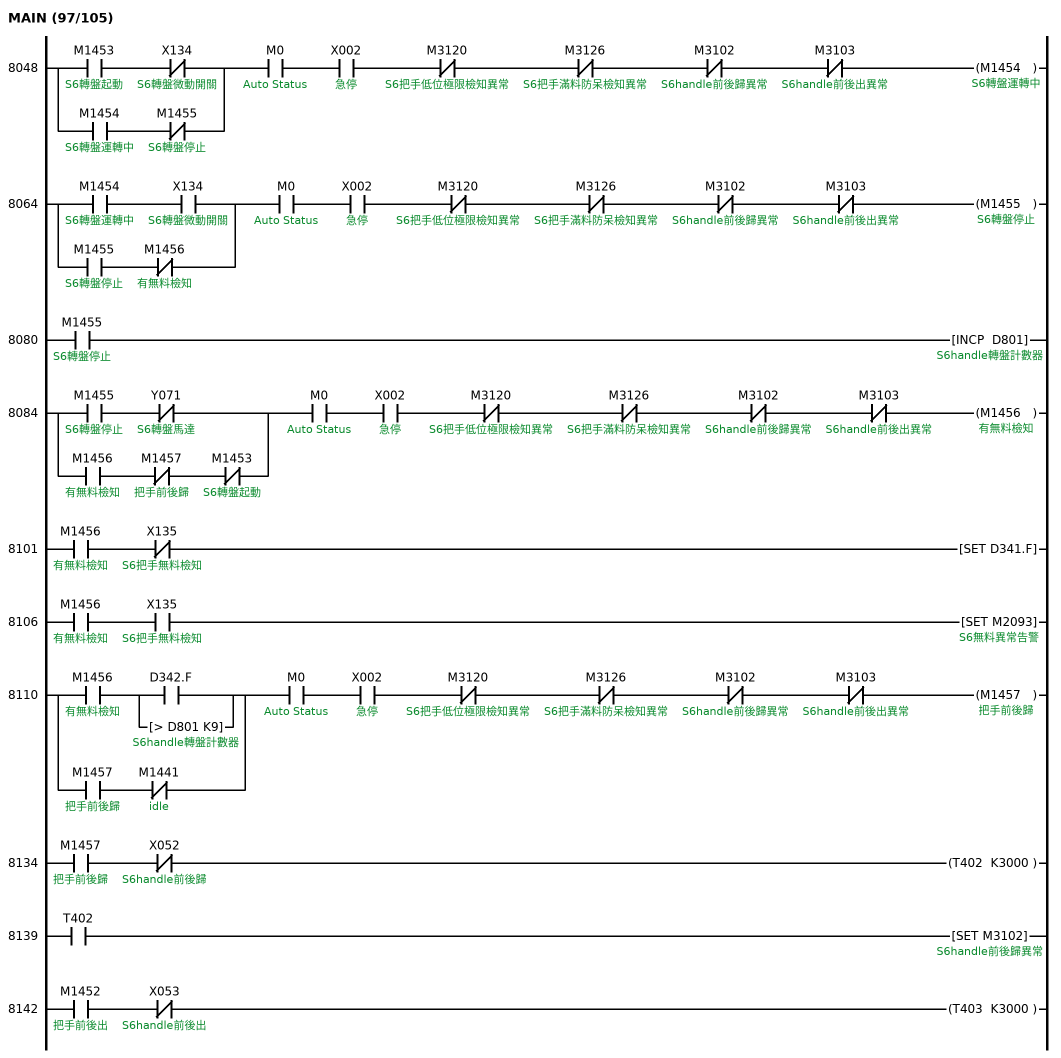
[picture p96: ladder of MAIN, rungs at steps 8048 to 8142]
8048  LD      M1453  ; S6轉盤起動
      ANI     X134  ; S6轉盤微動開關
      LD      M1454  ; S6轉盤運轉中
      ANI     M1455  ; S6轉盤停止
      ORB
      AND     M0  ; Auto Status
      AND     X002  ; 急停
      ANI     M3120  ; S6把手低位極限檢知異常
      ANI     M3126  ; S6把手滿料防呆檢知異常
      ANI     M3102  ; S6handle前後歸異常
      ANI     M3103  ; S6handle前後出異常
      OUT     M1454  ; S6轉盤運轉中
8064  LD      M1454  ; S6轉盤運轉中
      AND     X134  ; S6轉盤微動開關
      LD      M1455  ; S6轉盤停止
      ANI     M1456  ; 有無料檢知
      ORB
      AND     M0  ; Auto Status
      AND     X002  ; 急停
      ANI     M3120  ; S6把手低位極限檢知異常
      ANI     M3126  ; S6把手滿料防呆檢知異常
      ANI     M3102  ; S6handle前後歸異常
      ANI     M3103  ; S6handle前後出異常
      OUT     M1455  ; S6轉盤停止
8080  LD      M1455  ; S6轉盤停止
      INCP    D801
8084  LD      M1455  ; S6轉盤停止
      ANI     Y071  ; S6轉盤馬達
      LD      M1456  ; 有無料檢知
      ANI     M1457  ; 把手前後歸
      ANI     M1453  ; S6轉盤起動
      ORB
      AND     M0  ; Auto Status
      AND     X002  ; 急停
      ANI     M3120  ; S6把手低位極限檢知異常
      ANI     M3126  ; S6把手滿料防呆檢知異常
      ANI     M3102  ; S6handle前後歸異常
      ANI     M3103  ; S6handle前後出異常
      OUT     M1456  ; 有無料檢知
8101  LD      M1456  ; 有無料檢知
      ANI     X135  ; S6把手無料檢知
      SET     D341.F
8106  LD      M1456  ; 有無料檢知
      AND     X135  ; S6把手無料檢知
      SET     M2093  ; S6無料異常告警
8110  LD      M1456  ; 有無料檢知
      LD      D342.F
      OR>     D801 K9  ; S6handle轉盤計數器
      ANB
      LD      M1457  ; 把手前後歸
      ANI     M1441  ; idle
      ORB
      AND     M0  ; Auto Status
      AND     X002  ; 急停
      ANI     M3120  ; S6把手低位極限檢知異常
      ANI     M3126  ; S6把手滿料防呆檢知異常
      ANI     M3102  ; S6handle前後歸異常
      ANI     M3103  ; S6handle前後出異常
      OUT     M1457  ; 把手前後歸
8134  LD      M1457  ; 把手前後歸
      ANI     X052  ; S6handle前後歸
      OUT     T402 K3000
8139  LD      T402
      SET     M3102  ; S6handle前後歸異常
8142  LD      M1452  ; 把手前後出
      ANI     X053  ; S6handle前後出
      OUT     T403 K3000
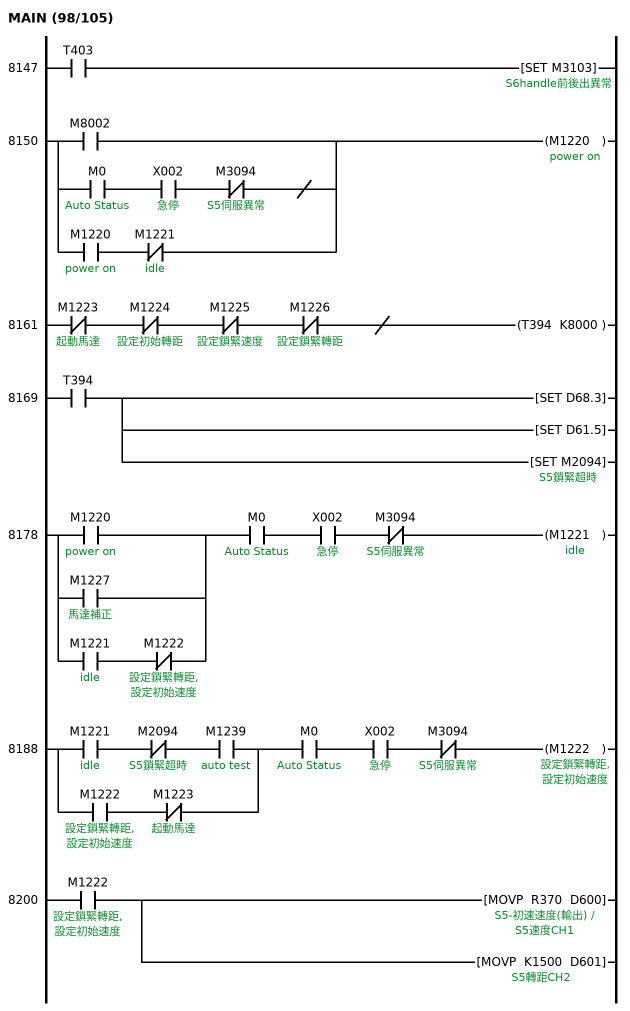
8147  LD      T403
      SET     M3103  ; S6handle前後出異常
8150  LD      M8002
      LD      M0  ; Auto Status
      AND     X002  ; 急停
      ANI     M3094  ; S5伺服異常
      INV
      ORB
      LD      M1220  ; power on
      ANI     M1221  ; idle
      ORB
      OUT     M1220  ; power on
8161  LDI     M1223  ; 起動馬達
      ANI     M1224  ; 設定初始轉距
      ANI     M1225  ; 設定鎖緊速度
      ANI     M1226  ; 設定鎖緊轉距
      INV
      OUT     T394 K8000
8169  LD      T394
      SET     D68.3
      SET     D61.5
      SET     M2094  ; S5鎖緊超時
8178  LD      M1220  ; power on
      OR      M1227  ; 馬達補正
      LD      M1221  ; idle
      ANI     M1222  ; 設定鎖緊轉距,設定初始速度
      ORB
      AND     M0  ; Auto Status
      AND     X002  ; 急停
      ANI     M3094  ; S5伺服異常
      OUT     M1221  ; idle
8188  LD      M1221  ; idle
      ANI     M2094  ; S5鎖緊超時
      AND     M1239  ; auto test
      LD      M1222  ; 設定鎖緊轉距,設定初始速度
      ANI     M1223  ; 起動馬達
      ORB
      AND     M0  ; Auto Status
      AND     X002  ; 急停
      ANI     M3094  ; S5伺服異常
      OUT     M1222  ; 設定鎖緊轉距,設定初始速度
8200  LD      M1222  ; 設定鎖緊轉距,設定初始速度
      MOVP    R370 D600
      MOVP    K1500 D601  ; S5轉距CH2
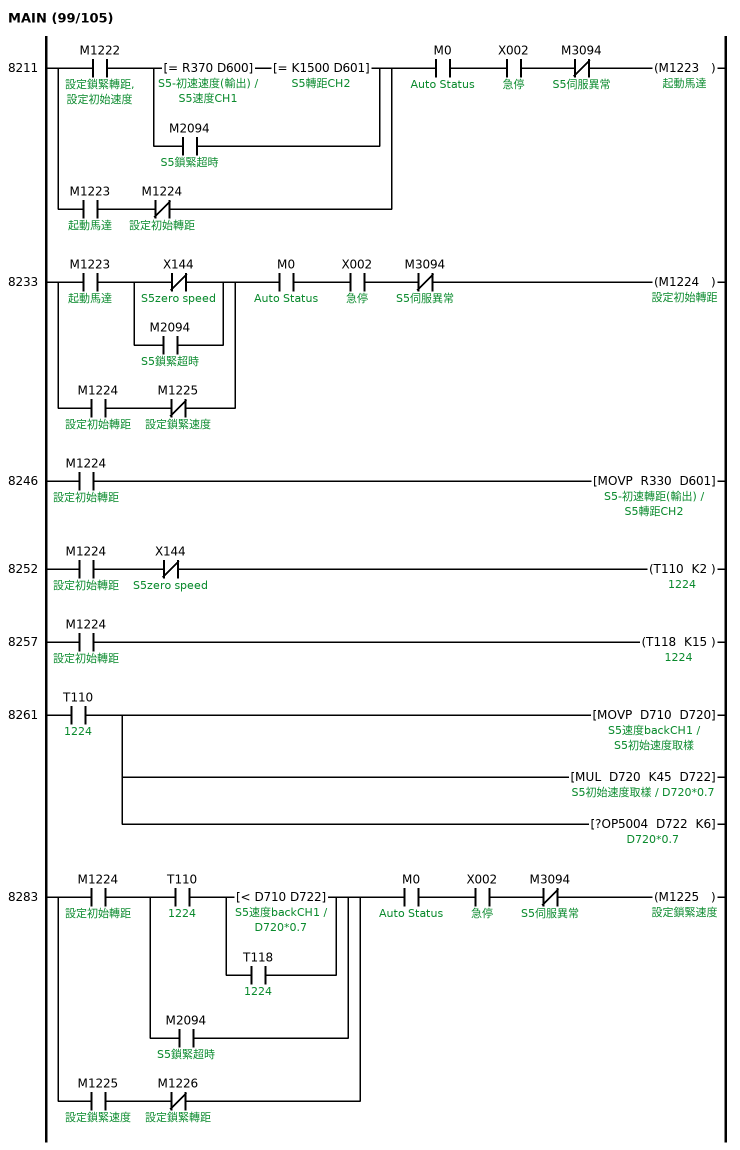
8211  LD      M1222  ; 設定鎖緊轉距,設定初始速度
      LD=     R370 D600  ; S5-初速速度(輸出) / S5速度CH1
      AND=    K1500 D601  ; S5轉距CH2
      OR      M2094  ; S5鎖緊超時
      ANB
      LD      M1223  ; 起動馬達
      ANI     M1224  ; 設定初始轉距
      ORB
      AND     M0  ; Auto Status
      AND     X002  ; 急停
      ANI     M3094  ; S5伺服異常
      OUT     M1223  ; 起動馬達
8233  LD      M1223  ; 起動馬達
      LDI     X144  ; S5zero speed
      OR      M2094  ; S5鎖緊超時
      ANB
      LD      M1224  ; 設定初始轉距
      ANI     M1225  ; 設定鎖緊速度
      ORB
      AND     M0  ; Auto Status
      AND     X002  ; 急停
      ANI     M3094  ; S5伺服異常
      OUT     M1224  ; 設定初始轉距
8246  LD      M1224  ; 設定初始轉距
      MOVP    R330 D601
8252  LD      M1224  ; 設定初始轉距
      ANI     X144  ; S5zero speed
      OUT     T110 K2  ; 1224
8257  LD      M1224  ; 設定初始轉距
      OUT     T118 K15  ; 1224
8261  LD      T110  ; 1224
      MOVP    D710 D720  ; S5初始速度取樣
      MUL     D720 K45 D722  ; D720*0.7
      ?OP5004 D722 K6
8283  LD      M1224  ; 設定初始轉距
      LD      T110  ; 1224
      LD<     D710 D722  ; S5速度backCH1 / D720*0.7
      OR      T118  ; 1224
      ANB
      OR      M2094  ; S5鎖緊超時
      ANB
      LD      M1225  ; 設定鎖緊速度
      ANI     M1226  ; 設定鎖緊轉距
      ORB
      AND     M0  ; Auto Status
      AND     X002  ; 急停
      ANI     M3094  ; S5伺服異常
      OUT     M1225  ; 設定鎖緊速度
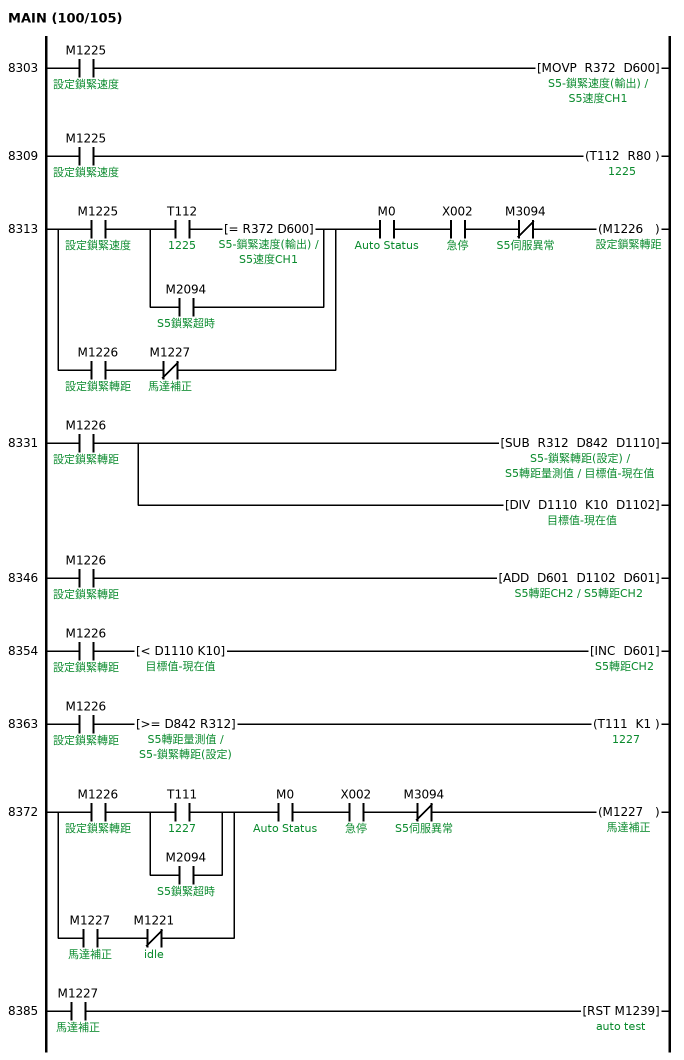
8303  LD      M1225  ; 設定鎖緊速度
      MOVP    R372 D600
8309  LD      M1225  ; 設定鎖緊速度
      OUT     T112 R80  ; 1225
8313  LD      M1225  ; 設定鎖緊速度
      LD      T112  ; 1225
      AND=    R372 D600  ; S5-鎖緊速度(輸出) / S5速度CH1
      OR      M2094  ; S5鎖緊超時
      ANB
      LD      M1226  ; 設定鎖緊轉距
      ANI     M1227  ; 馬達補正
      ORB
      AND     M0  ; Auto Status
      AND     X002  ; 急停
      ANI     M3094  ; S5伺服異常
      OUT     M1226  ; 設定鎖緊轉距
8331  LD      M1226  ; 設定鎖緊轉距
      SUB     R312 D842 D1110  ; 目標值-現在值
      DIV     D1110 K10 D1102
8346  LD      M1226  ; 設定鎖緊轉距
      ADD     D601 D1102 D601
8354  LD      M1226  ; 設定鎖緊轉距
      AND<    D1110 K10  ; 目標值-現在值
      INC     D601
8363  LD      M1226  ; 設定鎖緊轉距
      AND>=   D842 R312  ; S5轉距量測值 / S5-鎖緊轉距(設定)
      OUT     T111 K1  ; 1227
8372  LD      M1226  ; 設定鎖緊轉距
      LD      T111  ; 1227
      OR      M2094  ; S5鎖緊超時
      ANB
      LD      M1227  ; 馬達補正
      ANI     M1221  ; idle
      ORB
      AND     M0  ; Auto Status
      AND     X002  ; 急停
      ANI     M3094  ; S5伺服異常
      OUT     M1227  ; 馬達補正
8385  LD      M1227  ; 馬達補正
      RST     M1239  ; auto test
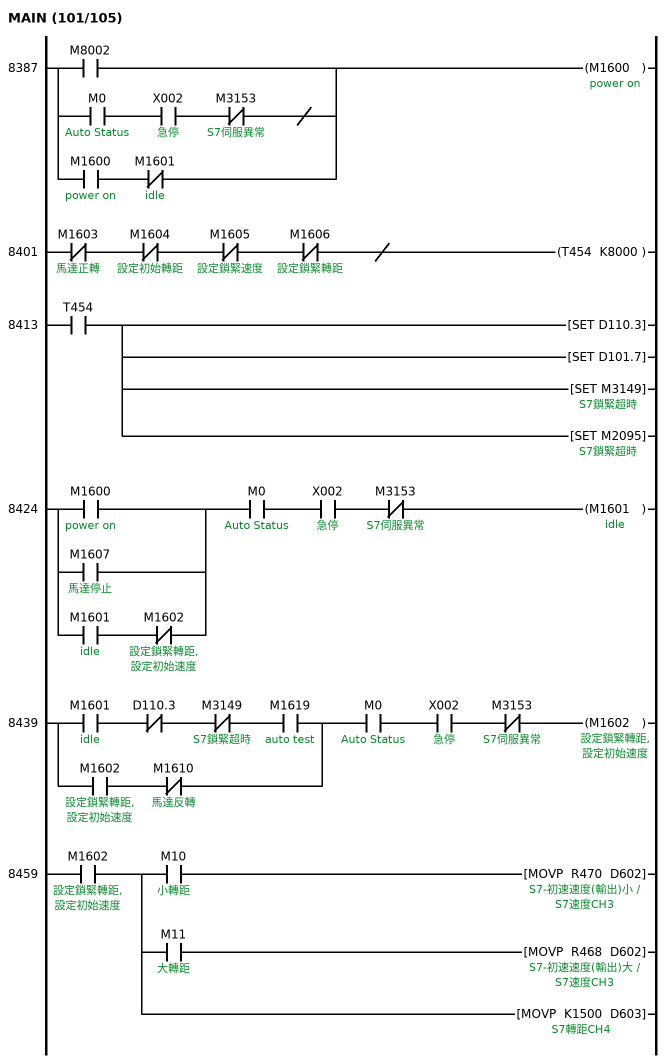
8387  LD      M8002
      LD      M0  ; Auto Status
      AND     X002  ; 急停
      ANI     M3153  ; S7伺服異常
      INV
      ORB
      LD      M1600  ; power on
      ANI     M1601  ; idle
      ORB
      OUT     M1600  ; power on
8401  LDI     M1603  ; 馬達正轉
      ANI     M1604  ; 設定初始轉距
      ANI     M1605  ; 設定鎖緊速度
      ANI     M1606  ; 設定鎖緊轉距
      INV
      OUT     T454 K8000
8413  LD      T454
      SET     D110.3
      SET     D101.7
      SET     M3149  ; S7鎖緊超時
      SET     M2095  ; S7鎖緊超時
8424  LD      M1600  ; power on
      OR      M1607  ; 馬達停止
      LD      M1601  ; idle
      ANI     M1602  ; 設定鎖緊轉距,設定初始速度
      ORB
      AND     M0  ; Auto Status
      AND     X002  ; 急停
      ANI     M3153  ; S7伺服異常
      OUT     M1601  ; idle
8439  LD      M1601  ; idle
      ANI     D110.3
      ANI     M3149  ; S7鎖緊超時
      AND     M1619  ; auto test
      LD      M1602  ; 設定鎖緊轉距,設定初始速度
      ANI     M1610  ; 馬達反轉
      ORB
      AND     M0  ; Auto Status
      AND     X002  ; 急停
      ANI     M3153  ; S7伺服異常
      OUT     M1602  ; 設定鎖緊轉距,設定初始速度
8459  LD      M1602  ; 設定鎖緊轉距,設定初始速度
      MPS
      AND     M10  ; 小轉距
      MOVP    R470 D602
      MRD
      AND     M11  ; 大轉距
      MOVP    R468 D602
      MPP
      MOVP    K1500 D603
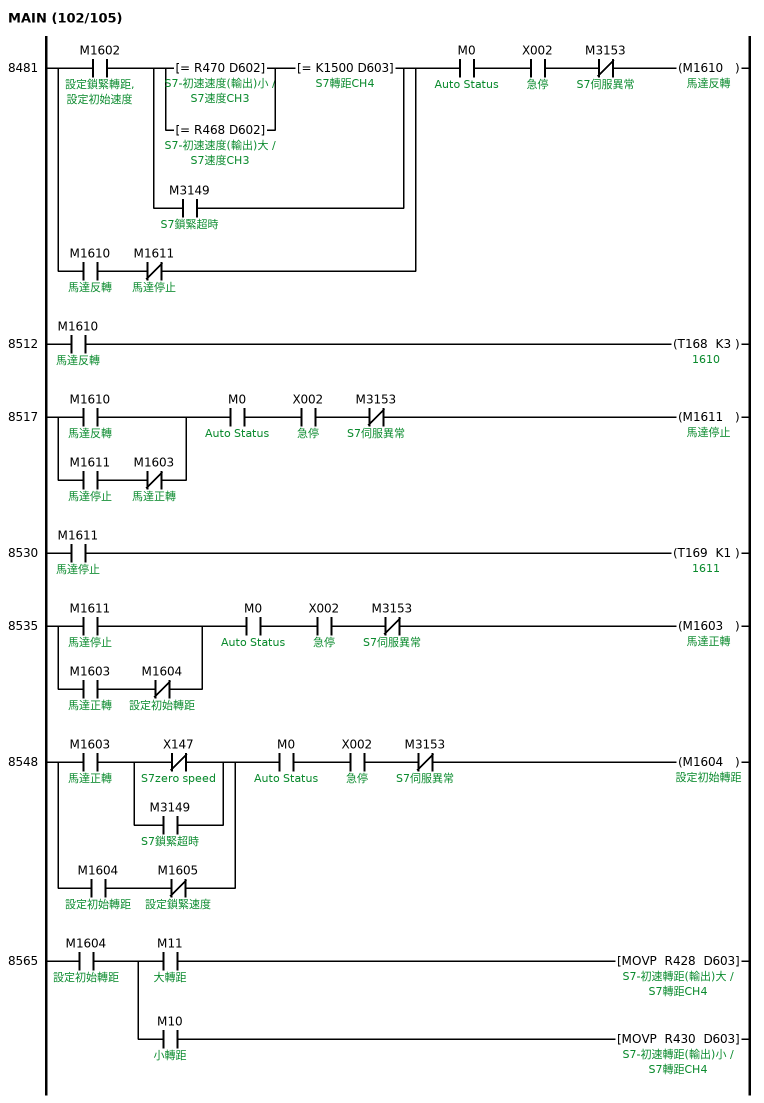
8481  LD      M1602  ; 設定鎖緊轉距,設定初始速度
      LD=     R470 D602  ; S7-初速速度(輸出)小 / S7速度CH3
      OR=     R468 D602  ; S7-初速速度(輸出)大 / S7速度CH3
      AND=    K1500 D603  ; S7轉距CH4
      OR      M3149  ; S7鎖緊超時
      ANB
      LD      M1610  ; 馬達反轉
      ANI     M1611  ; 馬達停止
      ORB
      AND     M0  ; Auto Status
      AND     X002  ; 急停
      ANI     M3153  ; S7伺服異常
      OUT     M1610  ; 馬達反轉
8512  LD      M1610  ; 馬達反轉
      OUT     T168 K3  ; 1610
8517  LD      M1610  ; 馬達反轉
      LD      M1611  ; 馬達停止
      ANI     M1603  ; 馬達正轉
      ORB
      AND     M0  ; Auto Status
      AND     X002  ; 急停
      ANI     M3153  ; S7伺服異常
      OUT     M1611  ; 馬達停止
8530  LD      M1611  ; 馬達停止
      OUT     T169 K1  ; 1611
8535  LD      M1611  ; 馬達停止
      LD      M1603  ; 馬達正轉
      ANI     M1604  ; 設定初始轉距
      ORB
      AND     M0  ; Auto Status
      AND     X002  ; 急停
      ANI     M3153  ; S7伺服異常
      OUT     M1603  ; 馬達正轉
8548  LD      M1603  ; 馬達正轉
      LDI     X147  ; S7zero speed
      OR      M3149  ; S7鎖緊超時
      ANB
      LD      M1604  ; 設定初始轉距
      ANI     M1605  ; 設定鎖緊速度
      ORB
      AND     M0  ; Auto Status
      AND     X002  ; 急停
      ANI     M3153  ; S7伺服異常
      OUT     M1604  ; 設定初始轉距
8565  LD      M1604  ; 設定初始轉距
      MPS
      AND     M11  ; 大轉距
      MOVP    R428 D603
      MPP
      AND     M10  ; 小轉距
      MOVP    R430 D603
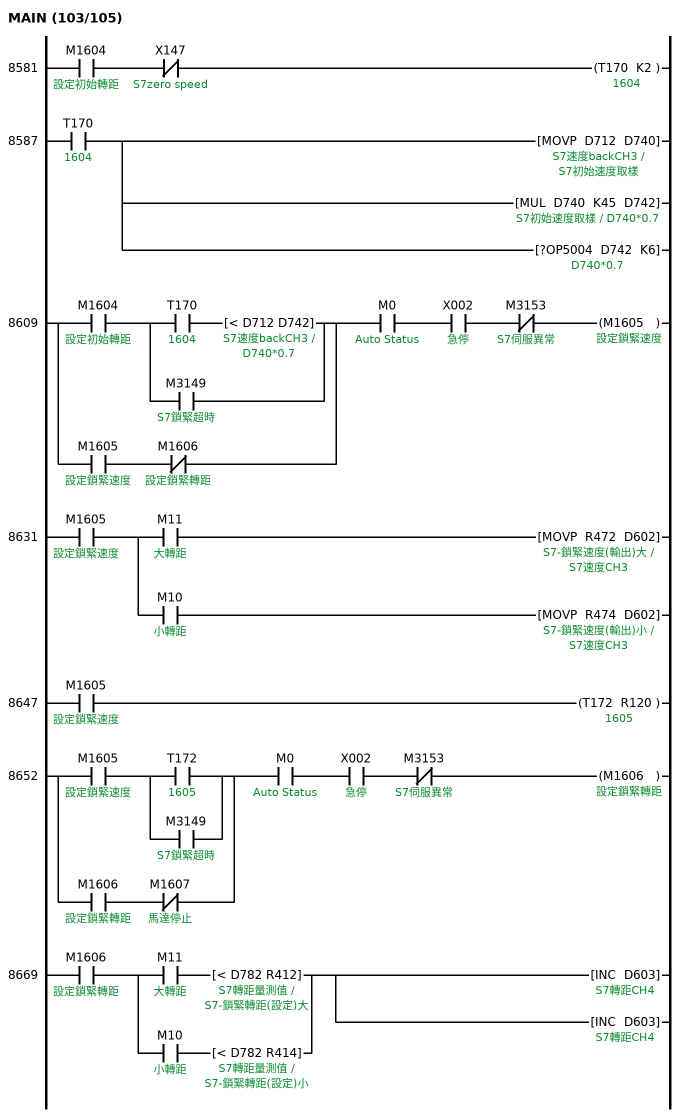
8581  LD      M1604  ; 設定初始轉距
      ANI     X147  ; S7zero speed
      OUT     T170 K2  ; 1604
8587  LD      T170  ; 1604
      MOVP    D712 D740  ; S7速度backCH3 / S7初始速度取樣
      MUL     D740 K45 D742  ; D740*0.7
      ?OP5004 D742 K6
8609  LD      M1604  ; 設定初始轉距
      LD      T170  ; 1604
      AND<    D712 D742  ; S7速度backCH3 / D740*0.7
      OR      M3149  ; S7鎖緊超時
      ANB
      LD      M1605  ; 設定鎖緊速度
      ANI     M1606  ; 設定鎖緊轉距
      ORB
      AND     M0  ; Auto Status
      AND     X002  ; 急停
      ANI     M3153  ; S7伺服異常
      OUT     M1605  ; 設定鎖緊速度
8631  LD      M1605  ; 設定鎖緊速度
      MPS
      AND     M11  ; 大轉距
      MOVP    R472 D602
      MPP
      AND     M10  ; 小轉距
      MOVP    R474 D602
8647  LD      M1605  ; 設定鎖緊速度
      OUT     T172 R120  ; 1605
8652  LD      M1605  ; 設定鎖緊速度
      LD      T172  ; 1605
      OR      M3149  ; S7鎖緊超時
      ANB
      LD      M1606  ; 設定鎖緊轉距
      ANI     M1607  ; 馬達停止
      ORB
      AND     M0  ; Auto Status
      AND     X002  ; 急停
      ANI     M3153  ; S7伺服異常
      OUT     M1606  ; 設定鎖緊轉距
8669  LD      M1606  ; 設定鎖緊轉距
      LD      M11  ; 大轉距
      AND<    D782 R412  ; S7轉距量測值 / S7-鎖緊轉距(設定)大
      LD      M10  ; 小轉距
      AND<    D782 R414  ; S7轉距量測值 / S7-鎖緊轉距(設定)小
      ORB
      ANB
      INC     D603
      INC     D603
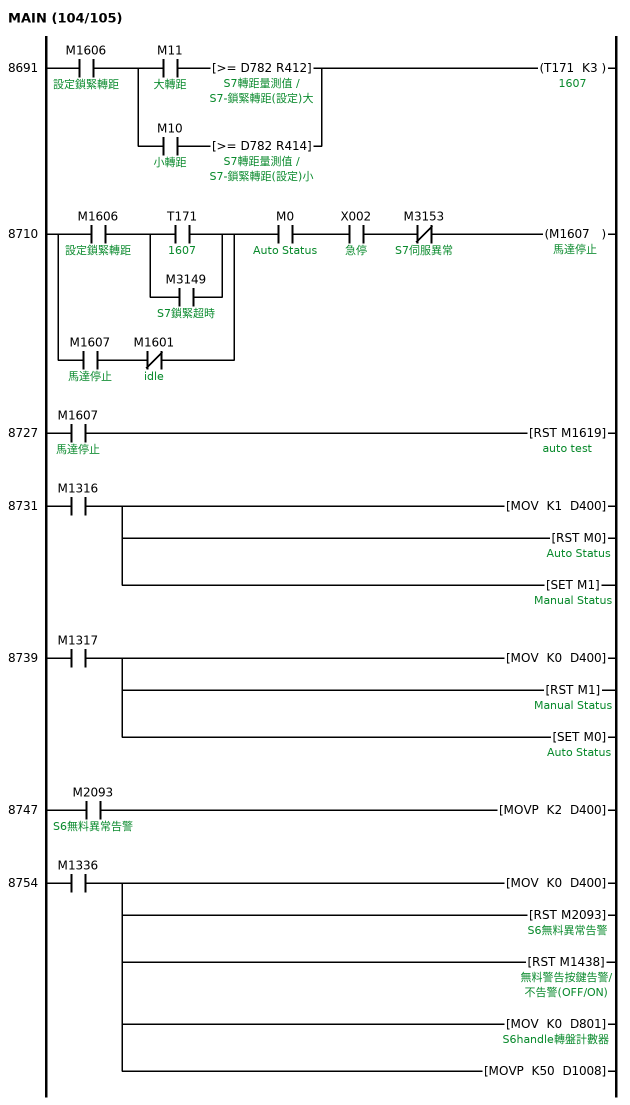
8691  LD      M1606  ; 設定鎖緊轉距
      LD      M11  ; 大轉距
      AND>=   D782 R412  ; S7轉距量測值 / S7-鎖緊轉距(設定)大
      LD      M10  ; 小轉距
      AND>=   D782 R414  ; S7轉距量測值 / S7-鎖緊轉距(設定)小
      ORB
      ANB
      OUT     T171 K3  ; 1607
8710  LD      M1606  ; 設定鎖緊轉距
      LD      T171  ; 1607
      OR      M3149  ; S7鎖緊超時
      ANB
      LD      M1607  ; 馬達停止
      ANI     M1601  ; idle
      ORB
      AND     M0  ; Auto Status
      AND     X002  ; 急停
      ANI     M3153  ; S7伺服異常
      OUT     M1607  ; 馬達停止
8727  LD      M1607  ; 馬達停止
      RST     M1619  ; auto test
8731  LD      M1316
      MOV     K1 D400
      RST     M0  ; Auto Status
      SET     M1  ; Manual Status
8739  LD      M1317
      MOV     K0 D400
      RST     M1  ; Manual Status
      SET     M0  ; Auto Status
8747  LD      M2093  ; S6無料異常告警
      MOVP    K2 D400
8754  LD      M1336
      MOV     K0 D400
      RST     M2093  ; S6無料異常告警
      RST     M1438  ; 無料警告按鍵告警/不告警(OFF/ON)
      MOV     K0 D801
      MOVP    K50 D1008
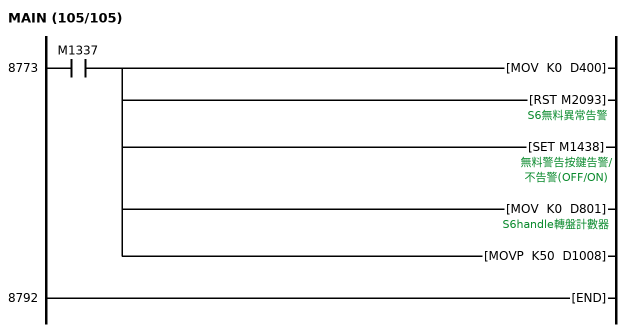
8773  LD      M1337
      MOV     K0 D400
      RST     M2093  ; S6無料異常告警
      SET     M1438  ; 無料警告按鍵告警/不告警(OFF/ON)
      MOV     K0 D801
      MOVP    K50 D1008
8792  END
END_PROGRAM

// device comments not shown above
M2  ; 停機/不停機(ON/OFF)
M569  ; S6轉盤動作完成flag
M570  ; 統計清除
M602  ; S2伺服RESETPB
M759  ; 無料flag
M1228  ; 馬達停止
M3001  ; S6轉盤微動開關異常
M3022  ; S2工件檢知異常
M3053  ; S3夾持料異常
M3092  ; S5浮鎖檢知異常
M3098  ; S5夾持料異常
M3121  ; S6把手高位極限檢知異常
M3125  ; S6把手無料檢知異常
M3150  ; S7浮鎖檢知異常
D1  ; #2NG狀態
D2  ; #2動作狀態
D5  ; #2第2站QC
D6  ; #2第3站QC
D7  ; #2第4站QC
D8  ; #2第5站QC
D9  ; #2第6站QC
D10  ; #2第7站QC
D11  ; #2第8站QC
D20  ; #3完成狀態
D21  ; #3NG狀態
D22  ; #3動作狀態
D25  ; #3第2站QC
D26  ; #3第3站QC
D27  ; #3第4站QC
D28  ; #3第5站QC
D29  ; #3第6站QC
D30  ; #3第7站QC
D31  ; #3第8站QC
D40  ; #4完成狀態
D41  ; #4NG狀態
D42  ; #4動作狀態
D45  ; #4第2站QC
D46  ; #4第3站QC
D47  ; #4第4站QC
D48  ; #4第5站QC
D49  ; #4第6站QC
D50  ; #4第7站QC
D51  ; #4第8站QC
D60  ; #5完成狀態
D61  ; #5NG狀態
D62  ; #5動作狀態
D63  ; #5放料完成
D65  ; #5第2站QC
D66  ; #5第3站QC
D67  ; #5第4站QC
D68  ; #5第5站QC
D69  ; #5第6站QC
D70  ; #5第7站QC
D71  ; #5第8站QC
D80  ; #6完成狀態
D81  ; #6NG狀態
D82  ; #6動作狀態
D83  ; #6放料完成
D85  ; #6第2站QC
D86  ; #6第3站QC
D87  ; #6第4站QC
D88  ; #6第5站QC
D89  ; #6第6站QC
D90  ; #6第7站QC
D91  ; #6第8站QC
D100  ; #7完成狀態
D101  ; #7NG狀態
D102  ; #7動作狀態
D103  ; #7放料完成
D105  ; #7第2站QC
D106  ; #7第3站QC
D107  ; #7第4站QC
D108  ; #7第5站QC
D109  ; #7第6站QC
D110  ; #7第7站QC
D111  ; #7第8站QC
D121  ; #8NG狀態
D122  ; #8動作狀態
D126  ; #8第3站QC
D128  ; #8第5站QC
D130  ; #8第7站QC
D140  ; #1完成狀態
D141  ; #1NG狀態
D142  ; #1動作狀態
D145  ; #1第2站QC
D146  ; #1第3站QC
D147  ; #1第4站QC
D148  ; #1第5站QC
D149  ; #1第6站QC
D150  ; #1第7站QC
D151  ; #1第8站QC
D510  ; *******
D701  ; CH2
D702  ; CH3
D703  ; CH4
D900  ; S6第1站狀態
D901  ; S6第2站狀態
D902  ; S6第3站狀態
D903  ; S6第4站狀態
D904  ; S6第5站狀態
D905  ; S6第6站狀態
D906  ; S6第7站狀態
D907  ; S6第8站狀態
R224  ; R222+R302
R226  ; R224*R304
R3001  ; #2NG狀態
R3002  ; #2動作狀態
R3005  ; #2第2站QC
R3006  ; #2第3站QC
R3007  ; #2第4站QC
R3008  ; #2第5站QC
R3009  ; #2第6站QC
R3010  ; #2第7站QC
R3011  ; #2第8站QC
R3012  ; #2第9站QC
R3013  ; #2第10站QC
R3014  ; #2第11站QC
R3015  ; #2第12站QC
R3016  ; #2第13站QC
R3017  ; #2第14站QC
R3018  ; #2第15站QC
R3019  ; #2第16站QC
T30  ; S2伺服起動
